{attribute 'qualified_only'}
{attribute 'strict'}
TYPE E_Station2_State :
(
		//GENERIC
	ABORTED				:=10,
	RESET_ERROR			:=20,
	HOMING				:=30,
	READY				:=40,
	//MANUAL_MODE			:=50, /manual mode not needed.
	ERROR				:=60,
	PERSISTENT_ERROR	:=70,
	STOPPING			:=80,
	//SPECIFIC FOR EVERY STATION
	MOVEMENT_A			:=100,
	MOVEMENT_B			:=120,
	MOVEMENT_C			:=130,
	DONE				:=140
);
END_TYPE

(* stored: Version 1.1.0.1, ProductVersion 3.1.4024.13
   DUT E_Station2_State: Id {5ddfb4d9-7fc1-463c-94a3-7a2a15a0ec39} *)
